// TIA Portal V20 export
TYPE "typeEmRelationShip"
// stored: Access Published, Namespace Unit1
   STRUCT
      General { ExternalAccessible := 'False'; ExternalVisible := 'False'; ExternalWritable := 'False'; S7_SetPoint := 'True'} : "Unit1.typeEmRelationshipParameters";
      EM0 { ExternalAccessible := 'False'; ExternalVisible := 'False'; ExternalWritable := 'False'; S7_SetPoint := 'True'} : "Unit1.typeEmRelationshipParameters";
      EM1 { ExternalAccessible := 'False'; ExternalVisible := 'False'; ExternalWritable := 'False'; S7_SetPoint := 'True'} : "Unit1.typeEmRelationshipParameters";
      EM2 { ExternalAccessible := 'False'; ExternalVisible := 'False'; ExternalWritable := 'False'; S7_SetPoint := 'True'} : "Unit1.typeEmRelationshipParameters";
      EM3 { ExternalAccessible := 'False'; ExternalVisible := 'False'; ExternalWritable := 'False'; S7_SetPoint := 'True'} : "Unit1.typeEmRelationshipParameters";
      EM4 { ExternalAccessible := 'False'; ExternalVisible := 'False'; ExternalWritable := 'False'; S7_SetPoint := 'True'} : "Unit1.typeEmRelationshipParameters";
      EM5 { ExternalAccessible := 'False'; ExternalVisible := 'False'; ExternalWritable := 'False'; S7_SetPoint := 'True'} : "Unit1.typeEmRelationshipParameters";
      EM6 { ExternalAccessible := 'False'; ExternalVisible := 'False'; ExternalWritable := 'False'; S7_SetPoint := 'True'} : "Unit1.typeEmRelationshipParameters";
      EM7 { ExternalAccessible := 'False'; ExternalVisible := 'False'; ExternalWritable := 'False'; S7_SetPoint := 'True'} : "Unit1.typeEmRelationshipParameters";
   END_STRUCT;
   // // EM0."Bool"[3] : RadiousMeasureReachedWarningLimit
   // // EM0.Data[21] : SepaUnwinderRadious
   // // EM1."Bool"[3] : RadiousMeasureReachedWarningLimit
   // // EM1.Data[21] : SepaUnwinderRadious
   // // EM2."Bool"[50] : OutPut_DancerPneumaticRegulatorReduceRequst
   // // EM2."Bool"[51] : OutPut_TopUnwinderRewindingRequset
   // // EM2."Bool"[52] : OutPut_BottomUnwinderRewindingRequset
   // // EM3."Bool"[21] : DancerPneumaticRegulatorReduceDone
   // // EM3."Bool"[22] : SepaFeedingRollerDownDone
   // // EM3."Bool"[23] : LoadCellTenstionDone
   // // EM3.Data[21] : CurrentDancerAngle
   // // EM4."Bool"[3] : mainPnp1Released
   // // EM4."Bool"[4] : mainPnp2Released
   // // EM4."Bool"[50] : OutPut_mainPnp1Released
   // // EM4."Bool"[51] : OutPut_mainPnp2Released
   // // EM4."Bool"[52] : OutPut_needToCell
   // // EM6.Data[0] : FinalRoller Anode Stack Pos
   // // EM6.Data[1] : FinalRoller Cathode Stack Pos
END_TYPE
